TYPE DUT_SERVER_SKILL_INPUT :
STRUCT
	///Range of parameters
	ParameterInput: DUT_SERVER_PARAMETERINPUTARRAY;
	///Start process
	Execute: BOOL;
END_STRUCT
END_TYPE

(* stored: Version 1.1.0.1, ProductVersion 3.1.0.25
   DUT DUT_SERVER_SKILL_INPUT: Id {ffc3cfd1-2d9f-4898-85a4-f3a1738ef16f} *)
